FUNCTION_BLOCK FB_Object_Testing
VAR_INPUT
	Start			: BOOL;
	Complete_test	: BOOL := FALSE;	
	RPDO_Nr			: BYTE := 0;
	TPDO_Nr			: BYTE := 0;
END_VAR
VAR_IN_OUT
	CAN_Object		: ST_CAN_Object;	
END_VAR
VAR_OUTPUT
	Finished		: BOOL := FALSE;	
END_VAR
VAR
	State			: INT := 0;
	i				: BYTE;
	
	Data			: ARRAY [0..255] OF BYTE;	
	SDO_READ		: FB_SDO_READ;
	SDO_WRITE		: FB_SDO_WRITE;
	
	Message			: STRING(128);
END_VAR

IF Start AND State = 255 THEN 
	Finished 	:= FALSE;
	State 		:= 0;
END_IF


SDO_READ(StartReading:=FALSE);
SDO_WRITE(StartWriting:=FALSE);


CASE State OF	
	// ************** Init **************	
	0:	// Init
		IF Start THEN
			IF CAN_Object.Length_Tested THEN 
				CAN_Object.Length_Tested := FALSE;
				CAN_Object.Length_Error := 0;
			ELSE
				CAN_Object.Length_Target := CAN_Object.Length; 
			END_IF
			
			IF CAN_Object.Readable_Tested THEN 
				CAN_Object.Readable_Tested := FALSE;
				CAN_Object.Readable_Error := 0;
				CAN_Object.Read_Value := 0;
			ELSE
				CAN_Object.Readable_Target := CAN_Object.Readable;
			END_IF
			
			IF CAN_Object.Writable_Tested THEN 
				CAN_Object.Writable_Tested := FALSE;
				CAN_Object.Writable_Error := 0; 
			ELSE		
				CAN_Object.Writable_Target := CAN_Object.Writable;
			END_IF
					
			IF CAN_Object.RPDO_Mappable_Tested THEN 
				CAN_Object.RPDO_Mappable_Tested := FALSE;
				CAN_Object.RPDO_Mappable_Error := 0; 
			ELSE		
				CAN_Object.RPDO_Mappable_Target := CAN_Object.RPDO_Mappable;
			END_IF
			
			IF CAN_Object.TPDO_Mappable_Tested THEN 
				CAN_Object.TPDO_Mappable_Tested := FALSE;
				CAN_Object.TPDO_Mappable_Error := 0; 
			ELSE		
				CAN_Object.TPDO_Mappable_Target := CAN_Object.TPDO_Mappable;
			END_IF			
			
			Message := 'Check "';
			Message := CONCAT(Message, CAN_Object.Name);
			Message := CONCAT(Message, '" (0x');
			Message := CONCAT(Message, WORD_TO_HEXSTR(CAN_Object.Index, 4, FALSE));
			Message := CONCAT(Message, ', ');
			Message := CONCAT(Message, BYTE_TO_STRING(CAN_Object.SubIndex));
			Message := CONCAT(Message, ', ');
			Message := CONCAT(Message, BYTE_TO_STRING(CAN_Object.Length * 8));
			Message := CONCAT(Message, ' bits)');
				
			GLB.Logger(Message:=Message);
			
			State := State + 1;
		END_IF
		
		
	// ******* Read and write test ******	
	1:	// Read Test
		IF CAN_Object.Readable_Target OR Complete_Test THEN			
			SDO_READ(
				ADSNetID		:= GLB.ADSNetID_CAN,				
				PortNr 		 	:= 16#1000 + GLB.NodeID,
				CO_Index 		:= CAN_Object.Index,
				CO_SubIndex 	:= CAN_Object.Subindex,
				DataLength 		:= CAN_Object.Length_Target,
				ReadData		=> Data,
				StartReading	:= TRUE	);		
			State := State + 1;
		ELSE				
			State := State + 10;
		END_IF
			
	2: // Read test, wait for finish
		IF SDO_READ.ReadDataAvailable THEN
			CAN_Object.Readable_Tested := TRUE;
			CAN_Object.Readable_Error := SDO_READ.Error;
			CAN_Object.Readable := (CAN_Object.Readable_Error = 0);
			
			Message := 'Reading: ';
			IF CAN_Object.Readable = CAN_Object.Readable_Target THEN
				Message := CONCAT(Message, 'OK');
				IF CAN_Object.Readable THEN
					Message := CONCAT(Message, ' / readable');
				ELSE
					Message := CONCAT(Message, ' / not readable');						
				END_IF
			ELSE
				Message := CONCAT(Message, 'Error');	
				IF CAN_Object.Readable THEN
					Message := CONCAT(Message, ' / should not be readable');
				ELSE
					Message := CONCAT(Message, ' / should be readable');						
				END_IF	
			END_IF	
			GLB.Logger(Message:=Message);
			
			IF CAN_Object.Readable THEN			
				CAN_Object.Read_Value := SHL(BYTE_TO_DWORD(SDO_READ.ReadData[3]),24) + SHL(BYTE_TO_DWORD(SDO_READ.ReadData[2]),16) + SHL(BYTE_TO_DWORD(SDO_READ.ReadData[1]),8) + BYTE_TO_DWORD(SDO_READ.ReadData[0]);
	
				// If Reading is successful, the length is also correct.
				CAN_Object.Length_Tested := TRUE;	
				CAN_Object.Length := CAN_Object.Length_Target;
				CAN_Object.Length_Error := 0;								
			END_IF
								
			State := State + 9;
		END_IF
	
		
	11:	// Write Test
		IF CAN_Object.Writable_Target OR Complete_Test THEN
			// Use the read value for write value?
			IF CAN_Object.Write_Value_Usage THEN CAN_Object.Write_Value := CAN_Object.Read_Value; END_IF
			
			FOR i := 0 TO CAN_Object.Length - 1 DO
				Data[i] := DWORD_TO_BYTE(SHR(CAN_Object.Write_Value, (8*i)));			
			END_FOR;
			
			SDO_WRITE(
				ADSNetID	:= GLB.ADSNetID_CAN,
				PortNr 		 := 16#1000 + GLB.NodeID,
				CO_Index 	 := CAN_Object.Index,
				CO_SubIndex  := CAN_Object.Subindex,
				DataLength 	 := CAN_Object.Length_Target,
				WriteData 	 := Data,
				StartWriting := TRUE );		
			State := State + 1;
		ELSE
			State := State + 10;
		END_IF
		
	12: // Write test, wait for finish
		IF SDO_WRITE.WriteDataFinished THEN
			CAN_Object.Writable_Tested := TRUE;
			CAN_Object.Writable_Error := SDO_WRITE.Error;
			CAN_Object.Writable := (CAN_Object.Writable_Error = 0);

			Message := 'Writing: ';
			IF CAN_Object.Writable = CAN_Object.Writable_Target THEN
				Message := CONCAT(Message, 'OK');
				IF CAN_Object.Writable THEN
					Message := CONCAT(Message, ' / writable');
				ELSE
					Message := CONCAT(Message, ' / not writable');						
				END_IF
			ELSE
				Message := CONCAT(Message, 'Error');	
				IF CAN_Object.Writable THEN
					Message := CONCAT(Message, ' / should be not writable');
				ELSE
					Message := CONCAT(Message, ' / should be writable');						
				END_IF
			END_IF	
			GLB.Logger(Message:=Message);					
	
			IF CAN_Object.Writable THEN
				CAN_Object.Write_Value := SHL(BYTE_TO_DWORD(SDO_Write.WriteData[3]),24) + SHL(BYTE_TO_DWORD(SDO_Write.WriteData[2]),16) + SHL(BYTE_TO_DWORD(SDO_Write.WriteData[1]),8) + BYTE_TO_DWORD(SDO_Write.WriteData[0]);				
				
				// If Writing is successful, the length is also correct.
				CAN_Object.Length_Tested := TRUE;
				CAN_Object.Length := CAN_Object.Length_Target;			
				CAN_Object.Length_Error := 0;						
			END_IF
		
			State := State + 9;				
		END_IF
		
		
	21: // Analyse the readable and writable tests
			// The PDO tests make only sense, if the object exists. This means that it must be readable and/or writable.
			IF CAN_Object.Readable OR CAN_Object.Writable THEN
				// Go to PDO tests
				State := 101;
			ELSE	
				IF Complete_test THEN
					// Additional tests
					i := 1;
					State := State + 1;
				ELSE
					// Test is finished with error.
					State := 254;					
				END_IF					
			END_IF
		
	
	22: // Redo the read test with other length
		SDO_READ(
			ADSNetID		:= GLB.ADSNetID_CAN,				
			PortNr 		 	:= 16#1000 + GLB.NodeID,
			CO_Index 		:= CAN_Object.Index,
			CO_SubIndex 	:= CAN_Object.Subindex,
			DataLength 		:= i,
			ReadData		=> Data,
			StartReading	:= TRUE	);		
		State := State + 1;	
		
	23: // Read test, wait for finish
		IF SDO_READ.ReadDataAvailable THEN
			CAN_Object.Readable_Tested := TRUE;
			CAN_Object.Readable_Error := SDO_READ.Error;
			CAN_Object.Readable := (CAN_Object.Readable_Error = 0);
						
			IF CAN_Object.Readable THEN
				CAN_Object.Read_Value := SHL(BYTE_TO_DWORD(SDO_READ.ReadData[3]),24) + SHL(BYTE_TO_DWORD(SDO_READ.ReadData[2]),16) + SHL(BYTE_TO_DWORD(SDO_READ.ReadData[1]),8) + BYTE_TO_DWORD(SDO_READ.ReadData[0]);	

				// If Reading is successful, the correct length is found.
				CAN_Object.Length_Tested := TRUE;	
				CAN_Object.Length := i;
				IF i > CAN_Object.Length_Target THEN			
					CAN_Object.Length_Error := 16#06070012;	
					CAN_Object.Readable_Error := 16#06070012;					
				ELSIF i < CAN_Object.Length_Target THEN
					CAN_Object.Length_Error := 16#06070013;	
					CAN_Object.Readable_Error := 16#06070013;				
				END_IF
				
				State := State + 1;
				
			ELSE					
				// This length is also wrong, check next length or resume with write test
				CASE i OF	
					1:
						IF (CAN_Object.Length_Target = 2) THEN
							// next length is 4 byte							
							i := 4;
							State := State - 1;							
						ELSE
							// next length is 2 byte							
							i := 2;
							State := State - 1;	
						END_IF
						
					2:
						IF (CAN_Object.Length_Target = 4) THEN
							// Continue with write test
							i := 1;
							State := State + 1;
						ELSE
							// next length is 4 byte
							i := 4;
							State := State - 1;	
						END_IF						
	
					4:
						// Continue with write test
						i := 1;
						State := State + 1;
						
					ELSE
						// If i value is strange, continue with write test
						i := 1;						
						State := State + 1;		
				END_CASE					
			END_IF		
		END_IF

		
	24: // Redo the write test with other length
		SDO_WRITE(
			ADSNetID	:= GLB.ADSNetID_CAN,
			PortNr 		 := 16#1000 + GLB.NodeID,
			CO_Index 	 := CAN_Object.Index,
			CO_SubIndex  := CAN_Object.Subindex,
			DataLength 	 := i,
			WriteData 	 := Data,
			StartWriting := TRUE );		
		State := State + 1;	
		
	25: // Write test, wait for finish
		IF SDO_WRITE.WriteDataFinished THEN
			CAN_Object.Writable_Tested := TRUE;
			CAN_Object.Writable_Error := SDO_WRITE.Error;
			CAN_Object.Writable := (CAN_Object.Writable_Error = 0);
						
			IF CAN_Object.Writable THEN
				CAN_Object.Write_Value := SHL(BYTE_TO_DWORD(SDO_Write.WriteData[3]),24) + SHL(BYTE_TO_DWORD(SDO_Write.WriteData[2]),16) + SHL(BYTE_TO_DWORD(SDO_Write.WriteData[1]),8) + BYTE_TO_DWORD(SDO_Write.WriteData[0]);				
				
				// If Writing is successful, the length is also correct.
				CAN_Object.Length_Tested := TRUE;
				CAN_Object.Length := i;		

				IF i > CAN_Object.Length_Target THEN			
					IF (CAN_Object.Length_Error = 16#06070013) THEN CAN_Object.Length_Error := 16#06070010; ELSE CAN_Object.Length_Error := 16#06070012; END_IF	
					CAN_Object.Writable_Error := 16#06070012;					
				ELSIF i < CAN_Object.Length_Target THEN
					IF (CAN_Object.Length_Error = 16#06070012) THEN CAN_Object.Length_Error := 16#06070010; ELSE CAN_Object.Length_Error := 16#06070013; END_IF
					CAN_Object.Writable_Error := 16#06070013;				
				END_IF
				
				State := State + 1;
			ELSE					
				// This length is also wrong, check next length or resume with next step
				CASE i OF	
					1:
						IF (CAN_Object.Length_Target = 2) THEN
							// next length is 4 byte							
							i := 4;
							State := State - 1;	
						ELSE
							// next length is 2 byte							
							i := 2;
							State := State - 1;	
						END_IF
						
					2:
						IF (CAN_Object.Length_Target = 4) THEN
							// Continue with write test
							State := State + 1;
						ELSE
							// next length is 4 byte
							i := 4;
							State := State - 1;	
						END_IF						
	
					4:
						// Continue with write test
						State := State + 1;
						
					ELSE
						// If i value is strange, continue with write test
						i := 1;						
						State := State + 1;		
				END_CASE				
			END_IF		
		END_IF
	
		
	26: // If the object is now found, resume with the PDO tests. Otherwise the test is finished with error.
		IF CAN_Object.Readable OR CAN_Object.Writable THEN
			State := 101;	
		ELSE
			State := 254;
		END_IF	
		
		
	// *********** PDO Tests ************
	101: // RPDO test
		IF CAN_Object.RPDO_Mappable_Target OR Complete_Test THEN	
			Data[0] := CAN_Object.Length * 8;
			Data[1] := CAN_Object.SubIndex;
			Data[2] := DWORD_TO_BYTE(CAN_Object.Index);
			Data[3] := DWORD_TO_BYTE(SHR(CAN_Object.Index,8));
				
			SDO_WRITE(
				ADSNetID	:= GLB.ADSNetID_CAN,
				PortNr 		 := 16#1000 + GLB.NodeID,
				CO_Index 	 := 16#1600 + RPDO_Nr,
				CO_SubIndex  := 1,
				DataLength 	 := 4,
				StartWriting := TRUE,
				WriteData 	 := Data );	
			State := State + 1;
		ELSE			
			State := State + 10;
		END_IF
			
	102: // RPDO test, wait for finish
		IF SDO_WRITE.WriteDataFinished THEN
			CAN_Object.RPDO_Mappable_Tested := TRUE;
			CAN_Object.RPDO_Mappable_Error := SDO_WRITE.Error;
			CAN_Object.RPDO_Mappable := (CAN_Object.RPDO_Mappable_Error = 0);	
			
			Message := 'Mappable RPDO: ';
			IF CAN_Object.RPDO_Mappable = CAN_Object.RPDO_Mappable_Target THEN
				Message := CONCAT(Message, 'OK');
				IF CAN_Object.RPDO_Mappable THEN
					Message := CONCAT(Message, ' / mappable');
				ELSE
					Message := CONCAT(Message, ' / not mappable');						
				END_IF
			ELSE
				Message := CONCAT(Message, 'Error');	
				IF CAN_Object.RPDO_Mappable THEN
					Message := CONCAT(Message, ' / should be not mappable');
				ELSE
					Message := CONCAT(Message, ' / should be mappable');						
				END_IF
			END_IF	
			GLB.Logger(Message:=Message);								
		
			State := State + 9;
		END_IF	

				
	111: // TPDO test
		IF CAN_Object.RPDO_Mappable_Target OR Complete_Test THEN		
			Data[0] := CAN_Object.Length * 8;
			Data[1] := CAN_Object.SubIndex;
			Data[2] := DWORD_TO_BYTE(CAN_Object.Index);
			Data[3] := DWORD_TO_BYTE(SHR(CAN_Object.Index,8));
	 
			SDO_WRITE(
				ADSNetID	:= GLB.ADSNetID_CAN,
				PortNr 		 := 16#1000 + GLB.NodeID,
				CO_Index 	 := 16#1A00 + TPDO_Nr,
				CO_SubIndex  := 1,
				DataLength 	 := 4,
				StartWriting := TRUE,
				WriteData 	 := Data );				
			State := State + 1;
		ELSE
			State := 254;
		END_IF
			
	112: // TPDO test, wait for finish
		IF SDO_WRITE.WriteDataFinished THEN
			CAN_Object.TPDO_Mappable_Tested := TRUE;
			CAN_Object.TPDO_Mappable_Error := SDO_WRITE.Error;
			CAN_Object.TPDO_Mappable := (CAN_Object.TPDO_Mappable_Error = 0);	
				
			Message := 'Mappable TPDO: ';
			IF CAN_Object.TPDO_Mappable = CAN_Object.TPDO_Mappable_Target THEN
				Message := CONCAT(Message, 'OK');
				IF CAN_Object.TPDO_Mappable THEN
					Message := CONCAT(Message, ' / mappable');
				ELSE
					Message := CONCAT(Message, ' / not mappable');						
				END_IF
			ELSE
				Message := CONCAT(Message, 'Error');	
				IF CAN_Object.TPDO_Mappable THEN
					Message := CONCAT(Message, ' / should be not mappable');
				ELSE
					Message := CONCAT(Message, ' / should be mappable');						
				END_IF
			END_IF	
			GLB.Logger(Message:=Message);	
			
			State := 254;
		END_IF

		
	// ************ Finished ************	
	254: // Check error 
	IF (CAN_Object.Mandatory > 0) OR CAN_Object.Readable OR CAN_Object.Writable THEN
		CAN_Object.Error := ((CAN_Object.Readable <> CAN_Object.Readable_Target) OR (CAN_Object.Writable <> CAN_Object.Writable_Target) OR  
							(CAN_Object.RPDO_Mappable <> CAN_Object.RPDO_Mappable_Target) OR (CAN_Object.TPDO_Mappable <> CAN_Object.TPDO_Mappable_Target) OR
							(CAN_Object.Length <> CAN_Object.Length_Target));

		Message := 'Result: ';
		IF CAN_Object.Error THEN
			Message := CONCAT(Message, 'Error');
		ELSE				
			Message := CONCAT(Message, 'OK');
		END_IF	
		Message := CONCAT(Message, '$0A**********');		
		GLB.Logger(Message:=Message, SaveFlag:=TRUE);	
	ELSE
		// Optional object not exists
		Message := 'Result: OK / Optional object does not exist';	
		Message := CONCAT(Message, '$0A**********');		
		GLB.Logger(Message:=Message, SaveFlag:=TRUE);	
	
	END_IF
	
		Finished := TRUE;	
		State := 255;
		
	255: // Tests finished
		Finished := TRUE;	
	
	
	ELSE	
		State := 254;
		
END_CASE

END_FUNCTION_BLOCK

(* stored: Version 1.1.0.1, ProductVersion 3.1.4024.11
   POU FB_Object_Testing: Id {b786489c-8b6d-4a02-93be-6647e41b4447}, SpecialFunc None *)
